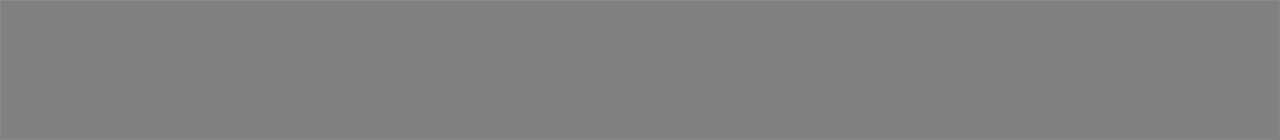
VISUALIZATION Header  // 1280x140
    Rectangle (0,0 1280x140)
END_VISUALIZATION

(* stored: Version 1.1.0.1, ProductVersion 3.1.4026.13
   Visu Header: Id {22b0bdeb-1fef-45d2-ac08-194fb2fab7cd} *)
